SUBAPPLICATION AUI_AUI_MUX_6_VAL (* 6-Wege-Multiplexer fuer AUI/UINT-Werte mit 6 internen initval_AUI und AUI_MUX_6 / AUI_AUI_MUX_6. Schaltet per Event-Input (EI1..EI6) zwischen val1..val6 um. *)
  (* Standard: 61499-2; Description: Copyright (c) 2026 Meisterschulen am Ostbahnhof This program and the accompanying materials are made available under the terms of the Eclipse Public License 2.0 which is available at https://www.eclipse.org/legal/epl-2.0/ SPDX-License-Identifier: EPL-2.0 *)
  (* Version 1.0, 2026-09-10, Franz Höpfinger, Meisterschulen am Ostbahnhof, 6-fach AUI/UINT MUX mit initval *)
  PACKAGE MyLib::sys;
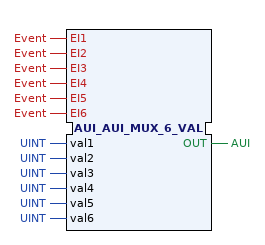
  EVENT_INPUT
    EI1; (* Event zur Auswahl von val1 *)
    EI2; (* Event zur Auswahl von val2 *)
    EI3; (* Event zur Auswahl von val3 *)
    EI4; (* Event zur Auswahl von val4 *)
    EI5; (* Event zur Auswahl von val5 *)
    EI6; (* Event zur Auswahl von val6 *)
  END_EVENT
  VAR_INPUT
    val1 : UINT; (* Initialer Ausgabewert bei EI1 *)
    val2 : UINT; (* Initialer Ausgabewert bei EI2 *)
    val3 : UINT; (* Initialer Ausgabewert bei EI3 *)
    val4 : UINT; (* Initialer Ausgabewert bei EI4 *)
    val5 : UINT; (* Initialer Ausgabewert bei EI5 *)
    val6 : UINT; (* Initialer Ausgabewert bei EI6 *)
  END_VAR
  PLUGS
    OUT : adapter::types::unidirectional::AUI; (* Ausgewaehlter AUI-Adapter Output *)
  END_PLUGS
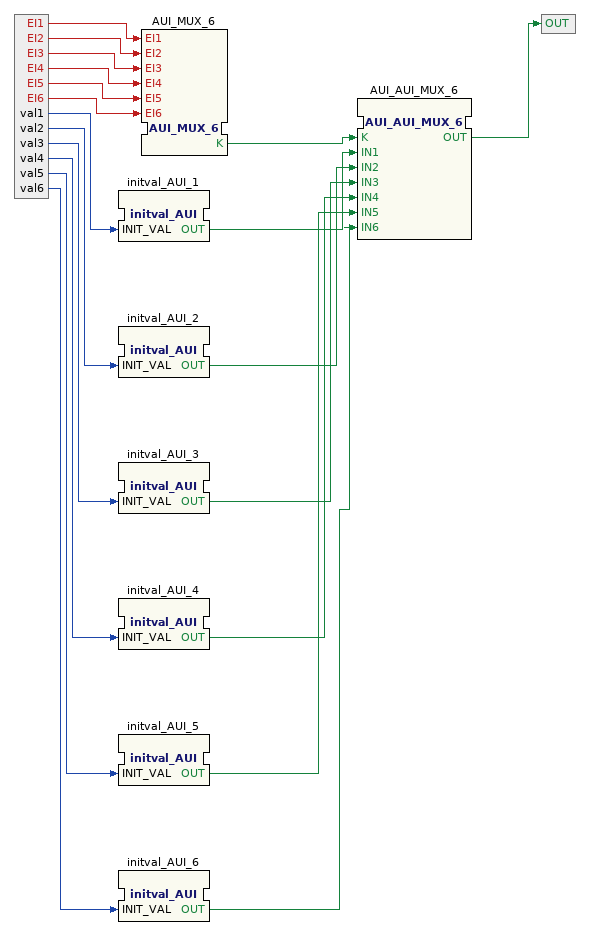
  FBS
    AUI_MUX_6 : adapter::events::unidirectional::AUI_MUX_6;
    AUI_AUI_MUX_6 : adapter::selection::unidirectional::AUI_AUI_MUX_6;
    initval_AUI_1 : adapter::types::unidirectional::AUI::initval::initval_AUI;
    initval_AUI_2 : adapter::types::unidirectional::AUI::initval::initval_AUI;
    initval_AUI_3 : adapter::types::unidirectional::AUI::initval::initval_AUI;
    initval_AUI_4 : adapter::types::unidirectional::AUI::initval::initval_AUI;
    initval_AUI_5 : adapter::types::unidirectional::AUI::initval::initval_AUI;
    initval_AUI_6 : adapter::types::unidirectional::AUI::initval::initval_AUI;
  END_FBS
  EVENT_CONNECTIONS
    EI1 TO AUI_MUX_6.EI1;
    EI2 TO AUI_MUX_6.EI2;
    EI3 TO AUI_MUX_6.EI3;
    EI4 TO AUI_MUX_6.EI4;
    EI5 TO AUI_MUX_6.EI5;
    EI6 TO AUI_MUX_6.EI6;
  END_CONNECTIONS
  DATA_CONNECTIONS
    val1 TO initval_AUI_1.INIT_VAL;
    val2 TO initval_AUI_2.INIT_VAL;
    val3 TO initval_AUI_3.INIT_VAL;
    val4 TO initval_AUI_4.INIT_VAL;
    val5 TO initval_AUI_5.INIT_VAL;
    val6 TO initval_AUI_6.INIT_VAL;
  END_CONNECTIONS
  ADAPTER_CONNECTIONS
    AUI_MUX_6.K TO AUI_AUI_MUX_6.K;
    initval_AUI_1.OUT TO AUI_AUI_MUX_6.IN1;
    initval_AUI_2.OUT TO AUI_AUI_MUX_6.IN2;
    initval_AUI_3.OUT TO AUI_AUI_MUX_6.IN3;
    initval_AUI_4.OUT TO AUI_AUI_MUX_6.IN4;
    initval_AUI_5.OUT TO AUI_AUI_MUX_6.IN5;
    initval_AUI_6.OUT TO AUI_AUI_MUX_6.IN6;
    AUI_AUI_MUX_6.OUT TO OUT;
  END_CONNECTIONS
END_SUBAPPLICATION
